Fanuc KAREL source: NC0040.KL

-- PROVISIONAL review KL for V1013-1; original PC SHA256 e9f042ff0a6bbe75ff41739c7ba4326e30b37a97a741674937280eb8104d9ccc
-- Incomplete behavior may be omitted. Consult companion uncertainty JSON. Do not deploy.
PROGRAM NC0040
%NOLOCKGROUP
-- UNRESOLVED_LOCAL_POOL 1 cells at code offset 3; source declarations unknown
-- DIRECT_LOCAL_WORD_ACCESS alone does not prove INTEGER, REAL, or BOOLEAN
BEGIN
  -- UNRESOLVED_PC offsets 0-8; opcodes 2B,2C,7B
  -- UNRESOLVED_PC offsets 13-20; opcodes 9D,23
  -- UNRESOLVED_PC offsets 25-42; opcodes 21,40,41,42
  -- UNRESOLVED_PC offsets 47-81; opcodes 21,2E,52,23,7A,40,41,42
  -- UNRESOLVED_PC offsets 86-110; opcodes 21,2E,52,23,7A,43
  -- UNRESOLVED_PC offsets 115-132; opcodes 21,40,41,42
  -- UNRESOLVED_PC offsets 137-171; opcodes 21,2E,52,23,7A,40,41,42
  -- UNRESOLVED_PC offsets 176-200; opcodes 21,2E,52,23,7A,43
  -- UNRESOLVED_PC offsets 205-222; opcodes 21,40,41,42
  -- UNRESOLVED_PC offsets 227-261; opcodes 21,2E,52,23,7A,40,41,42
  -- UNRESOLVED_PC offsets 266-290; opcodes 21,2E,52,23,7A,43
  -- UNRESOLVED_PC offsets 295-312; opcodes 21,40,41,42
  -- UNRESOLVED_PC offsets 317-351; opcodes 21,2E,52,23,7A,40,41,42
  -- UNRESOLVED_PC offsets 356-380; opcodes 21,2E,52,23,7A,43
  -- UNRESOLVED_PC offsets 385-402; opcodes 21,40,41,42
  -- UNRESOLVED_PC offsets 407-441; opcodes 21,2E,52,23,7A,40,41,42
  -- UNRESOLVED_PC offsets 446-470; opcodes 21,2E,52,23,7A,43
  -- UNRESOLVED_PC offsets 475-492; opcodes 21,40,41,42
  -- UNRESOLVED_PC offsets 497-531; opcodes 21,2E,52,23,7A,40,41,42
  -- UNRESOLVED_PC offsets 536-560; opcodes 21,2E,52,23,7A,43
  -- UNRESOLVED_PC offsets 565-582; opcodes 21,40,41,42
  -- UNRESOLVED_PC offsets 587-621; opcodes 21,2E,52,23,7A,40,41,42
  -- UNRESOLVED_PC offsets 626-650; opcodes 21,2E,52,23,7A,43
  -- UNRESOLVED_PC offsets 655-672; opcodes 21,40,41,42
  -- UNRESOLVED_PC offsets 677-711; opcodes 21,2E,52,23,7A,40,41,42
  -- UNRESOLVED_PC offsets 716-740; opcodes 21,2E,52,23,7A,43
  -- UNRESOLVED_PC offsets 745-762; opcodes 21,40,41,42
  -- UNRESOLVED_PC offsets 767-801; opcodes 21,2E,52,23,7A,40,41,42
  -- UNRESOLVED_PC offsets 806-830; opcodes 21,2E,52,23,7A,43
  -- UNRESOLVED_PC offsets 835-852; opcodes 21,40,41,42
  -- UNRESOLVED_PC offsets 857-891; opcodes 21,2E,52,23,7A,40,41,42
  -- UNRESOLVED_PC offsets 896-920; opcodes 21,2E,52,23,7A,43
  -- UNRESOLVED_PC offsets 925-942; opcodes 21,40,41,42
  -- UNRESOLVED_PC offsets 947-981; opcodes 21,2E,52,23,7A,40,41,42
  -- UNRESOLVED_PC offsets 986-1010; opcodes 21,2E,52,23,7A,43
  -- UNRESOLVED_PC offsets 1015-1032; opcodes 21,40,41,42
  -- UNRESOLVED_PC offsets 1037-1071; opcodes 21,2E,52,23,7A,40,41,42
  -- UNRESOLVED_PC offsets 1076-1100; opcodes 21,2E,52,23,7A,43
  -- UNRESOLVED_PC offsets 1105-1122; opcodes 21,40,41,42
  -- UNRESOLVED_PC offsets 1127-1161; opcodes 21,2E,52,23,7A,40,41,42
  -- UNRESOLVED_PC offsets 1166-1190; opcodes 21,2E,52,23,7A,43
  -- UNRESOLVED_PC offsets 1195-1212; opcodes 21,40,41,42
  -- UNRESOLVED_PC offsets 1217-1251; opcodes 21,2E,52,23,7A,40,41,42
  -- UNRESOLVED_PC offsets 1256-1280; opcodes 21,2E,52,23,7A,43
  -- UNRESOLVED_PC offsets 1285-1302; opcodes 21,40,41,42
  -- UNRESOLVED_PC offsets 1307-1341; opcodes 21,2E,52,23,7A,40,41,42
  -- UNRESOLVED_PC offsets 1346-1370; opcodes 21,2E,52,23,7A,43
  -- UNRESOLVED_PC offsets 1375-1392; opcodes 21,40,41,42
  -- UNRESOLVED_PC offsets 1397-1431; opcodes 21,2E,52,23,7A,40,41,42
  -- UNRESOLVED_PC offsets 1436-1460; opcodes 21,2E,52,23,7A,43
  -- UNRESOLVED_PC offsets 1465-1482; opcodes 21,40,41,42
  -- UNRESOLVED_PC offsets 1487-1521; opcodes 21,2E,52,23,7A,40,41,42
  -- UNRESOLVED_PC offsets 1526-1550; opcodes 21,2E,52,23,7A,43
  -- UNRESOLVED_PC offsets 1555-1572; opcodes 21,40,41,42
  -- UNRESOLVED_PC offsets 1577-1611; opcodes 21,2E,52,23,7A,40,41,42
  -- UNRESOLVED_PC offsets 1616-1640; opcodes 21,2E,52,23,7A,43
  -- UNRESOLVED_PC offsets 1645-1659; opcodes 21,9D,52,23
  -- UNRESOLVED_PC offsets 1754-1758; opcodes 7F
  -- UNRESOLVED_PC offsets 1763-1767; opcodes 27,AA
  -- UNRESOLVED_PC offsets 1772-1776; opcodes 7F
END NC0040
